(* IEC 61131-3 sources: programs/VI-54/VI-54_20171205/VI-54_20171205/Stations/PLC_VI54/VI-54_171014/Class/DiasDriveSplitter, 1 file *)

(* ---- DiasDriveSplitter.st ---- *)
(*!
<Class
	Name               = "DiasDriveSplitter"
	Revision           = "6.1"
	RealtimeTask       = "false"
	CyclicTask         = "true"
	BackgroundTask     = "false"
	Sigmatek           = "false"
	OSInterface        = "false"
	HighPriority       = "false"
	Automatic          = "false"
	UpdateMode         = "Prescan"
	SharedCommandTable = "true"
	Objectsize         = "(570,480)">
	<Channels>
		<Server Name="ClassSvr" Visualized="true" Initialize="false" WriteProtected="false" Retentive="false"/>
		<Server Name="DrivesEnabled" Visualized="true" Initialize="false" WriteProtected="true" Retentive="false"/>
		<Server Name="DrivesOk" Visualized="true" Initialize="false" WriteProtected="false" Retentive="false"/>
		<Client Name="DriveAxleM1" Required="true" Internal="false" Comment="Connected to the _DriveAxis&#13;&#10;"/>
		<Client Name="DriveAxleM2" Required="false" Internal="false" Comment="Connected to the _DriveAxis"/>
		<Client Name="DriveAxleM3" Required="false" Internal="false" Comment="Connected to the _DriveAxis"/>
		<Client Name="DriveAxleM4" Required="false" Internal="false" Comment="Connected to the _DriveAxis"/>
		<Client Name="DriveAxleM5" Required="false" Internal="false" Comment="Connected to the _DriveAxis"/>
		<Client Name="DriveAxleM6" Required="false" Internal="false" Comment="Connected to the _DriveAxis"/>
		<Client Name="DriveAxleM7" Required="false" Internal="false"/>
		<Client Name="DriveAxleM8" Required="false" Internal="false"/>
	</Channels>
	<Network Name="DiasDriveSplitter">
		<!-- List of Components in this network -->
		<Components>
		</Components>
		<Comments>
		</Comments>
		<!-- List of Connections in this network -->
		<Connections>
		</Connections>
		<!-- Headerfiles -->
		<Options>
		</Options>
	</Network>
</Class>
*)
DiasDriveSplitter : CLASS
  //Servers:
	ClassSvr 	: SvrChCmd_DINT;
	DrivesOk 	: SvrCh_DINT;
	DrivesEnabled 	: SvrCh_DINT;
  //Clients:
	DriveAxleM1 	: CltChCmd_DriveAxleErr;
	DriveAxleM2 	: CltChCmd_DriveAxleErr;
	DriveAxleM3 	: CltChCmd_DriveAxleErr;
	DriveAxleM4 	: CltChCmd_DriveAxleErr;
	DriveAxleM5 	: CltChCmd_DriveAxleErr;
	DriveAxleM6 	: CltChCmd_DriveAxleErr;
	DriveAxleM7 	: CltChCmd_DriveAxleErr;
	DriveAxleM8 	: CltChCmd_DriveAxleErr;
  //Variables:
		DriveManagerOnline 	: DINT;
		AxleOkM1 	: DINT;
		AxleOkM2 	: DINT;
		AxleOkM3 	: DINT;
		AxleOkM4 	: DINT;
		AxleOkM5 	: DINT;
		AxleOkM6 	: DINT;
		AxleOkM7 	: DINT;
		AxleOkM8 	: DINT;
		AxleEnableM1 	: DINT;
		AxleEnableM2 	: DINT;
		AxleEnableM3 	: DINT;
		AxleEnableM4 	: DINT;
		AxleEnableM5 	: DINT;
		AxleEnableM6 	: DINT;
		AxleEnableM7 	: DINT;
		AxleEnableM8 	: DINT;
		cmdResetDrives 	: DINT;
  //Functions:

	FUNCTION VIRTUAL GLOBAL CyWork
		VAR_INPUT
			EAX 	: UDINT;
		END_VAR
		VAR_OUTPUT
			state (EAX) 	: UDINT;
		END_VAR;

	FUNCTION GLOBAL ReadDriveOk
		VAR_OUTPUT
			State 	: DINT;
		END_VAR;

	FUNCTION GLOBAL ReadDrivesEnabled
		VAR_OUTPUT
			State 	: DINT;
		END_VAR;

	FUNCTION VIRTUAL GLOBAL DrivesOk::Write
		VAR_INPUT
			input (EAX) 	: DINT;
		END_VAR
		VAR_OUTPUT
			result (EAX) 	: DINT;
		END_VAR;
  //Tables:
	FUNCTION @STD
		VAR_OUTPUT
			ret_code	: CONFSTATES;
		END_VAR;
	FUNCTION GLOBAL TAB @CT_;
END_CLASS;

#pragma usingLtd DriveAxleErr

FUNCTION VIRTUAL GLOBAL DiasDriveSplitter::CyWork
	VAR_INPUT
		EAX 	: UDINT;
	END_VAR
	VAR_OUTPUT
		state (EAX) 	: UDINT;
	END_VAR

  // Axle number 1
  if IsClientConnected(#DriveAxleM1) then
    DriveAxleM1  := DriveAxleM1.Read();
    AxleOkM1     := DriveAxleM1.ReadDriveOk();
    AxleEnableM1 := DriveAxleM1.ReadDriveEnabled();
    if cmdResetDrives = 1 then
      DriveAxleM1.ResetDrives();
    end_if;
  else
    DriveAxleM1  := ERROR;
    AxleEnableM1 := 1; // Axle enabled
    AxleOkM1     := 1;// axle oke
  end_if;

  // Axle number 2
  if IsClientConnected(#DriveAxleM2) then
    DriveAxleM2  := DriveAxleM2.Read();
    AxleOkM2     := DriveAxleM2.ReadDriveOk();
    AxleEnableM2 := DriveAxleM2.ReadDriveEnabled();
    if cmdResetDrives = 1 then
      DriveAxleM2.ResetDrives();
    end_if;
  else
    DriveAxleM2  := ERROR;
    AxleEnableM2 := 1; // Axle enabled
    AxleOkM2     := 1;// axle oke
  end_if;

  // Axle number 3
  if IsClientConnected(#DriveAxleM3) then
    DriveAxleM3  := DriveAxleM3.Read();
    AxleOkM3     := DriveAxleM3.ReadDriveOk();
    AxleEnableM3 := DriveAxleM3.ReadDriveEnabled();
    if cmdResetDrives = 1 then
      DriveAxleM3.ResetDrives();
    end_if;
  else
    DriveAxleM3  := ERROR;
    AxleEnableM3 := 1; // Axle enabled
    AxleOkM3     := 1;// axle oke
  end_if;

  // Axle number 4
  if IsClientConnected(#DriveAxleM4) then
    DriveAxleM4  := DriveAxleM4.Read();
    AxleOkM4     := DriveAxleM4.ReadDriveOk();
    AxleEnableM4 := DriveAxleM4.ReadDriveEnabled();
    if cmdResetDrives = 1 then
      DriveAxleM4.ResetDrives();
    end_if;
  else
    DriveAxleM4  := ERROR;
    AxleEnableM4 := 1; // Axle enabled
    AxleOkM4     := 1;// axle oke
  end_if;

  // Axle number 5
  if IsClientConnected(#DriveAxleM5) then
    DriveAxleM5  := DriveAxleM5.Read();
    AxleOkM5     := DriveAxleM5.ReadDriveOk();
    AxleEnableM5 := DriveAxleM5.ReadDriveEnabled();
    if cmdResetDrives = 1 then
      DriveAxleM5.ResetDrives();
    end_if;
  else
    DriveAxleM5  := ERROR;
    AxleEnableM5 := 1; // Axle enabled
    AxleOkM5     := 1;// axle oke
  end_if;

  // Axle number 6
  if IsClientConnected(#DriveAxleM6) then
    DriveAxleM6  := DriveAxleM6.Read();
    AxleOkM6     := DriveAxleM6.ReadDriveOk();
    AxleEnableM6 := DriveAxleM6.ReadDriveEnabled();
    if cmdResetDrives = 1 then
      DriveAxleM6.ResetDrives();
    end_if;
  else
    DriveAxleM6  := ERROR;
    AxleEnableM6 := 1; // Axle enabled
    AxleOkM6     := 1;// axle oke
  end_if;

  // Axle number 7
  if IsClientConnected(#DriveAxleM7) then
    DriveAxleM7  := DriveAxleM7.Read();
    AxleOkM7     := DriveAxleM7.ReadDriveOk();
    AxleEnableM7 := DriveAxleM7.ReadDriveEnabled();
    if cmdResetDrives = 1 then
      DriveAxleM7.ResetDrives();
    end_if;
  else
    DriveAxleM7  := ERROR;
    AxleEnableM7 := 1; // Axle enabled
    AxleOkM7     := 1;// axle oke
  end_if;

  // Axle number 8
  if IsClientConnected(#DriveAxleM8) then
    DriveAxleM8  := DriveAxleM8.Read();
    AxleOkM8     := DriveAxleM8.ReadDriveOk();
    AxleEnableM8 := DriveAxleM8.ReadDriveEnabled();
    if cmdResetDrives = 1 then
      DriveAxleM8.ResetDrives();
    end_if;
  else
    DriveAxleM8  := ERROR;
    AxleEnableM8 := 1; // Axle enabled
    AxleOkM8     := 1;// axle oke
  end_if;

  DrivesEnabled := ((AxleEnableM1 = 1 & AxleEnableM2 = 1 & AxleEnableM3 = 1 & AxleEnableM4 = 1 & AxleEnableM5 = 1 & AxleEnableM6 = 1 & AxleEnableM7 = 1 & AxleEnableM8 = 1));
  DrivesOK      := ((AxleOkM1 = 1 & AxleOkM2 = 1 & AxleOkM3 = 1 & AxleOkM4 = 1 & AxleOkM5 = 1 & AxleOkM6 = 1 & AxleOkM7 = 1 & AxleOkM8 = 1));

	state := READY;

END_FUNCTION

FUNCTION GLOBAL DiasDriveSplitter::ReadDriveOk
	VAR_OUTPUT
		State 	: DINT;
	END_VAR

  State := DrivesOk;

END_FUNCTION

FUNCTION GLOBAL DiasDriveSplitter::ReadDrivesEnabled
	VAR_OUTPUT
		State 	: DINT;
	END_VAR

  State := DrivesEnabled;

END_FUNCTION

FUNCTION VIRTUAL GLOBAL DiasDriveSplitter::DrivesOk::Write
	VAR_INPUT
		input (EAX) 	: DINT;
	END_VAR
	VAR_OUTPUT
		result (EAX) 	: DINT;
	END_VAR

  if DrivesOk = 0 then
    cmdResetDrives := input;
  end_if;

 	result := input;

END_FUNCTION
